FUNCTION F_Contains : BOOL
VAR_INPUT
    s      : STRING;
    needle : STRING;
END_VAR

END_FUNCTION

(* stored: Version 1.1.0.1
   POU F_Contains: Id {83736892-b9f9-479f-8686-bbc3853ffa25}, SpecialFunc None *)
